FUNCTION TcoDintToBytes
VAR_INPUT
	inFormat : eTcoDataFormat;
	inValue : DINT;
END_VAR
VAR_IN_OUT
    outByte0: BYTE;
    outByte1: BYTE;
    outByte2: BYTE;
    outByte3: BYTE;
END_VAR
VAR
	_b0: BYTE;
	_b1: BYTE;
	_b2: BYTE;
    _b3: BYTE;

	_tmpDINT : DINT; 
END_VAR

_tmpDINT:=inValue;

_b3:=UDINT_TO_BYTE(_tmpDINT MOD 256);
_tmpDINT:=SHR(_tmpDINT,8);
_b2:=UDINT_TO_BYTE(_tmpDINT MOD 256);
_tmpDINT:=SHR(_tmpDINT,8);
_b1:=UDINT_TO_BYTE(_tmpDINT MOD 256);
_tmpDINT:=SHR(_tmpDINT,8);
_b0:=UDINT_TO_BYTE(_tmpDINT MOD 256);
_tmpDINT:=SHR(_tmpDINT,8);

IF inFormat=eTcoDataFormat.LittleEndian THEN
	outByte0 := _b3;
	outByte1 := _b2;	
	outByte2 := _b1;
	outByte3 := _b0;	
ELSIF inFormat=eTcoDataFormat.BigEndian THEN
	outByte0 := _b0;
	outByte1 := _b1;	
	outByte2 := _b2;
	outByte3 := _b3;	
END_IF

END_FUNCTION

(* stored: Version 1.1.0.1, ProductVersion 3.1.4024.12
   POU TcoDintToBytes: Id {3981a929-ee0b-4efd-ac82-5ebbcdc07710}, SpecialFunc None *)
